PROGRAM VISU
VAR
	posizioneProsciutto: INT;
	posizioneProsciuttoY: INT;
	rotazionePiattaforma: INT;
	prosciuttoVisibile: BOOL;
	Random: DRAND;
	PB1Trig: R_TRIG;
	SmistamentoTrig: F_TRIG;
END_VAR

Random(Seed:= 100); //Numero casuale
PB1Trig(CLK := GVL.PB1); //Fronte di salita del pulsante
SmistamentoTrig(CLK := MAIN.Smistamento); //Indica quando termina uno smistamento

//Reset posizione alla fine dello smistamento o alla pressione di Start
IF PB1Trig.Q OR SmistamentoTrig.Q THEN
	GVL.LC1 := Random.Num * 10;
	prosciuttoVisibile := TRUE;
	posizioneProsciutto := 0;
	posizioneProsciuttoY := 0;
	rotazionePiattaforma := 0;
	GVL.PS1 := 0;
END_IF

IF GVL.M1 THEN
	posizioneProsciutto := posizioneProsciutto +2;
END_IF

IF GVL.M5 AND rotazionePiattaforma = 0 THEN
	posizioneProsciutto := posizioneProsciutto +4;
END_IF

IF GVL.M5 AND rotazionePiattaforma = 90 THEN
	posizioneProsciuttoY := posizioneProsciuttoY +2;
END_IF

IF GVL.M5 AND rotazionePiattaforma = 270 THEN
	posizioneProsciuttoY := posizioneProsciuttoY -2;
END_IF

IF posizioneProsciutto >= 160 AND NOT MAIN.Smistamento THEN
	GVL.PS1 := TRUE;
ELSE
	GVL.PS1 := FALSE;
END_IF

IF posizioneProsciutto >= 350 THEN
	GVL.PS3 := TRUE;
	prosciuttoVisibile:= FALSE;
ELSE
	GVL.PS3 := FALSE;
END_IF

IF posizioneProsciuttoY >= 200 THEN
	GVL.PS2 := TRUE;
	prosciuttoVisibile:= FALSE;
ELSE
	GVL.PS2 := FALSE;
END_IF

IF posizioneProsciuttoY <= -200 THEN
	GVL.PS4 := TRUE;
	prosciuttoVisibile:= FALSE;
ELSE
	GVL.PS4 := FALSE;
END_IF



IF GVL.M4 THEN
	rotazionePiattaforma := rotazionePiattaforma +2;
	IF rotazionePiattaforma = 360 THEN
		rotazionePiattaforma := 0;
	END_IF
END_IF

CASE rotazionePiattaforma OF
	0:
		GVL.SB1 := TRUE;
		GVL.SB2 := FALSE;
		GVL.SB3 := FALSE;
	90:
		GVL.SB1 := FALSE;
		GVL.SB2 := TRUE;
		GVL.SB3 := FALSE;
	270:
		GVL.SB1 := FALSE;
		GVL.SB2 := FALSE;
		GVL.SB3 := TRUE;
	ELSE
		GVL.SB1 := FALSE;
		GVL.SB2 := FALSE;
		GVL.SB3 := FALSE;
END_CASE

END_PROGRAM

(* stored: Version 1.1.0.1, ProductVersion 3.1.4024.12
   POU VISU: Id {1338be45-51f0-44d8-871a-f3970fab8a28}, SpecialFunc None *)
